// TIA Portal V17 export
// export: Created 2021-12-03T08:13:06.5776488Z, ExportSetting WithDefaults, DisplayName Totally Integrated Automation Portal, DisplayVersion V17, DisplayName TIA Portal Openness, DisplayVersion V17, DisplayName TIA Portal Version Control Interface, DisplayVersion V17, DisplayName STEP 7 Professional, DisplayVersion V17, DisplayName STEP 7 Safety, DisplayVersion V17, DisplayName WinCC Advanced, DisplayVersion V17
DATA_BLOCK "DBI_SM_Conv"   // DB530
AUTHOR : MNi
VERSION : 0.1
// stored: AutoNumber false, InstanceOfName FB_SM_Conv, InstanceOfType FB
"FB_SM_Conv"
   // VAR_INPUT
   //    I_InitTrue : Bool;
   // END_VAR
   // VAR RETAIN
   //    S_State : Array[1..25] of Bool;
   //    S_Conditions : Array[1..30] of Bool;
   //    S_Actions_Out : Array[1..15] of Bool;
   //    S_Actions_Trans : Array[1..15] of Bool;
   //    S_Actions_In : Array[1..15] of Bool;
   //    S_ActState : Int;
   //    S_ActionAct_Out : Bool;
   //    S_ActionAct_Trans : Bool;
   //    S_ActionAct_In : Bool;
   //    S_Parameter : Struct
   //       AutoFastSpd : Int;
   //       AutoSlowSpd : Int;
   //       JoggSpd : Int;
   //       Ramp : Int;
   //    END_STRUCT;
   //    S_ControlCommand_In : Struct
   //       PrSSlowOpn : Bool;
   //       PrSSlowCls : Bool;
   //    END_STRUCT;
   //    S_ControlCommand_Out : Struct
   //       ReqSingleMode : Bool;
   //       MovingFwd : Bool;
   //       MovingBwrd : Bool;
   //       RefSpd : Int;
   //       Ramp : Int;
   //    END_STRUCT;
   //    S_HomingToOpn : Bool;
   // END_VAR
BEGIN
END_DATA_BLOCK
